(* IEC 61131-3 sources: SafePLC-Gen-Evaluation/Evaluation Results/eastman/run_03, 2 files *)

(* ---- io_declarations.st ---- *)
(* ==================================================  *)
(* PLC I/O Variable Declarations — CODESYS 3.5  *)
(* Generated by SafePLC-Gen Multimodal  *)
(* ==================================================  *)

VAR_GLOBAL
    (* --- Analog Inputs ---  *)
    FI_1_Raw                     AT %IW0       : INT := 0;    (* FI-1 — Flow indicator on feed line P-65 enterin  *)
    FI_2_Raw                     AT %IW2       : INT := 0;    (* FI-2 — Flow indicator on line P-54/P-53 associa  *)
    FI_3_Raw                     AT %IW4       : INT := 0;    (* FI-3 — Flow indicator on line P-57 associated w  *)
    TI_1_Raw                     AT %IW6       : INT := 0;    (* TI-1 — Temperature indicator TI-1, local panel   *)
    TI_4_Raw                     AT %IW8       : INT := 0;    (* TI-4 — Temperature indicator TI-4 on line P-12   *)
    TI_5_Raw                     AT %IW10      : INT := 0;    (* TI-5 — Temperature indicator TI-5 on line P-53   *)
    TI_6_Raw                     AT %IW12      : INT := 0;    (* TI-6 — Temperature indicator TI-6 on line assoc  *)
    TI_7_Raw                     AT %IW14      : INT := 0;    (* TI-7 — Temperature indicator TI-7 on line P-20/  *)
    TI_8_Raw                     AT %IW16      : INT := 0;    (* TI-8 — Temperature indicator TI-8 on line P-57   *)
    (* --- Analog Outputs ---  *)
    V_3_Out                      AT %QW0       : INT := 0;    (* V-3 — Control valve V-3 on line P-28 from Deca  *)
    V_4_Out                      AT %QW2       : INT := 0;    (* V-4 — Control valve V-4 on line P-74/P-12 feed  *)
    V_5_Out                      AT %QW4       : INT := 0;    (* V-5 — Control valve V-5 on line P-38/P-83 refl  *)
    V_7_Out                      AT %QW6       : INT := 0;    (* V-7 — Control valve V-7 on line P-19 vent or p  *)
END_VAR

(* ---- generated_code.st ---- *)
(* Generated by SafePLC-Gen Multimodal — CODESYS 3.5 *)
(* IEC 61131-3 Structured Text *)
(* Date: 2026-04-25T12:33:26.075096 *)

PROGRAM DistillationControl

VAR
    FI_1_Raw                     AT %IW0       : INT := 0;
    FI_2_Raw                     AT %IW2       : INT := 0;
    FI_3_Raw                     AT %IW4       : INT := 0;
    TI_1_Raw                     AT %IW6       : INT := 0;
    TI_4_Raw                     AT %IW8       : INT := 0;
    TI_5_Raw                     AT %IW10      : INT := 0;
    TI_6_Raw                     AT %IW12      : INT := 0;
    TI_7_Raw                     AT %IW14      : INT := 0;
    TI_8_Raw                     AT %IW16      : INT := 0;
    V_3_Out                      AT %QW0       : INT := 0;
    V_4_Out                      AT %QW2       : INT := 0;
    V_5_Out                      AT %QW4       : INT := 0;
    V_7_Out                      AT %QW6       : INT := 0;
END_VAR

VAR
    FirstScan                    : BOOL := TRUE;

    FI_1_Scaled                  : REAL := 0.0;
    FI_2_Scaled                  : REAL := 0.0;
    FI_3_Scaled                  : REAL := 0.0;
    TI_1_Scaled                  : REAL := 0.0;
    TI_4_Scaled                  : REAL := 0.0;
    TI_5_Scaled                  : REAL := 0.0;
    TI_6_Scaled                  : REAL := 0.0;
    TI_7_Scaled                  : REAL := 0.0;
    TI_8_Scaled                  : REAL := 0.0;

    FI_1_HH_SP                   : REAL := 180.0;
    FI_1_H_SP                    : REAL := 160.0;
    FI_1_L_SP                    : REAL := 40.0;
    FI_1_LL_SP                   : REAL := 20.0;
    FI_1_Deadband                : REAL := 2.0;
    FI_1_HH                      : BOOL := FALSE;
    FI_1_H                       : BOOL := FALSE;
    FI_1_L                       : BOOL := FALSE;
    FI_1_LL                      : BOOL := FALSE;
    FI_1_HH_Latch                : SR := (S1 := FALSE, R := FALSE);
    FI_1_LL_Latch                : SR := (S1 := FALSE, R := FALSE);
    FI_1_HH_Ack                  : BOOL := FALSE;
    FI_1_LL_Ack                  : BOOL := FALSE;

    FI_2_HH_SP                   : REAL := 180.0;
    FI_2_H_SP                    : REAL := 160.0;
    FI_2_L_SP                    : REAL := 40.0;
    FI_2_LL_SP                   : REAL := 20.0;
    FI_2_Deadband                : REAL := 2.0;
    FI_2_HH                      : BOOL := FALSE;
    FI_2_H                       : BOOL := FALSE;
    FI_2_L                       : BOOL := FALSE;
    FI_2_LL                      : BOOL := FALSE;
    FI_2_HH_Latch                : SR := (S1 := FALSE, R := FALSE);
    FI_2_LL_Latch                : SR := (S1 := FALSE, R := FALSE);
    FI_2_HH_Ack                  : BOOL := FALSE;
    FI_2_LL_Ack                  : BOOL := FALSE;

    FI_3_HH_SP                   : REAL := 180.0;
    FI_3_H_SP                    : REAL := 160.0;
    FI_3_L_SP                    : REAL := 40.0;
    FI_3_LL_SP                   : REAL := 20.0;
    FI_3_Deadband                : REAL := 2.0;
    FI_3_HH                      : BOOL := FALSE;
    FI_3_H                       : BOOL := FALSE;
    FI_3_L                       : BOOL := FALSE;
    FI_3_LL                      : BOOL := FALSE;
    FI_3_HH_Latch                : SR := (S1 := FALSE, R := FALSE);
    FI_3_LL_Latch                : SR := (S1 := FALSE, R := FALSE);
    FI_3_HH_Ack                  : BOOL := FALSE;
    FI_3_LL_Ack                  : BOOL := FALSE;

    TI_1_HH_SP                   : REAL := 120.0;
    TI_1_H_SP                    : REAL := 110.0;
    TI_1_L_SP                    : REAL := 30.0;
    TI_1_LL_SP                   : REAL := 20.0;
    TI_1_Deadband                : REAL := 1.0;
    TI_1_HH                      : BOOL := FALSE;
    TI_1_H                       : BOOL := FALSE;
    TI_1_L                       : BOOL := FALSE;
    TI_1_LL                      : BOOL := FALSE;
    TI_1_HH_Latch                : SR := (S1 := FALSE, R := FALSE);
    TI_1_LL_Latch                : SR := (S1 := FALSE, R := FALSE);
    TI_1_HH_Ack                  : BOOL := FALSE;
    TI_1_LL_Ack                  : BOOL := FALSE;

    TI_4_HH_SP                   : REAL := 120.0;
    TI_4_H_SP                    : REAL := 110.0;
    TI_4_L_SP                    : REAL := 30.0;
    TI_4_LL_SP                   : REAL := 20.0;
    TI_4_Deadband                : REAL := 1.0;
    TI_4_HH                      : BOOL := FALSE;
    TI_4_H                       : BOOL := FALSE;
    TI_4_L                       : BOOL := FALSE;
    TI_4_LL                      : BOOL := FALSE;
    TI_4_HH_Latch                : SR := (S1 := FALSE, R := FALSE);
    TI_4_LL_Latch                : SR := (S1 := FALSE, R := FALSE);
    TI_4_HH_Ack                  : BOOL := FALSE;
    TI_4_LL_Ack                  : BOOL := FALSE;

    TI_5_HH_SP                   : REAL := 120.0;
    TI_5_H_SP                    : REAL := 110.0;
    TI_5_L_SP                    : REAL := 30.0;
    TI_5_LL_SP                   : REAL := 20.0;
    TI_5_Deadband                : REAL := 1.0;
    TI_5_HH                      : BOOL := FALSE;
    TI_5_H                       : BOOL := FALSE;
    TI_5_L                       : BOOL := FALSE;
    TI_5_LL                      : BOOL := FALSE;
    TI_5_HH_Latch                : SR := (S1 := FALSE, R := FALSE);
    TI_5_LL_Latch                : SR := (S1 := FALSE, R := FALSE);
    TI_5_HH_Ack                  : BOOL := FALSE;
    TI_5_LL_Ack                  : BOOL := FALSE;

    TI_6_HH_SP                   : REAL := 120.0;
    TI_6_H_SP                    : REAL := 110.0;
    TI_6_L_SP                    : REAL := 30.0;
    TI_6_LL_SP                   : REAL := 20.0;
    TI_6_Deadband                : REAL := 1.0;
    TI_6_HH                      : BOOL := FALSE;
    TI_6_H                       : BOOL := FALSE;
    TI_6_L                       : BOOL := FALSE;
    TI_6_LL                      : BOOL := FALSE;
    TI_6_HH_Latch                : SR := (S1 := FALSE, R := FALSE);
    TI_6_LL_Latch                : SR := (S1 := FALSE, R := FALSE);
    TI_6_HH_Ack                  : BOOL := FALSE;
    TI_6_LL_Ack                  : BOOL := FALSE;

    TI_7_HH_SP                   : REAL := 120.0;
    TI_7_H_SP                    : REAL := 110.0;
    TI_7_L_SP                    : REAL := 30.0;
    TI_7_LL_SP                   : REAL := 20.0;
    TI_7_Deadband                : REAL := 1.0;
    TI_7_HH                      : BOOL := FALSE;
    TI_7_H                       : BOOL := FALSE;
    TI_7_L                       : BOOL := FALSE;
    TI_7_LL                      : BOOL := FALSE;
    TI_7_HH_Latch                : SR := (S1 := FALSE, R := FALSE);
    TI_7_LL_Latch                : SR := (S1 := FALSE, R := FALSE);
    TI_7_HH_Ack                  : BOOL := FALSE;
    TI_7_LL_Ack                  : BOOL := FALSE;

    TI_8_HH_SP                   : REAL := 120.0;
    TI_8_H_SP                    : REAL := 110.0;
    TI_8_L_SP                    : REAL := 30.0;
    TI_8_LL_SP                   : REAL := 20.0;
    TI_8_Deadband                : REAL := 1.0;
    TI_8_HH                      : BOOL := FALSE;
    TI_8_H                       : BOOL := FALSE;
    TI_8_L                       : BOOL := FALSE;
    TI_8_LL                      : BOOL := FALSE;
    TI_8_HH_Latch                : SR := (S1 := FALSE, R := FALSE);
    TI_8_LL_Latch                : SR := (S1 := FALSE, R := FALSE);
    TI_8_HH_Ack                  : BOOL := FALSE;
    TI_8_LL_Ack                  : BOOL := FALSE;

    V3_SP                        : REAL := 100.0;
    V3_Kp                        : REAL := 1.2;
    V3_Ki                        : REAL := 0.05;
    V3_Integral                  : REAL := 0.0;
    V3_Error                     : REAL := 0.0;
    V3_Output                    : REAL := 50.0;

    V4_SP                        : REAL := 80.0;
    V4_Kp                        : REAL := 1.5;
    V4_Ki                        : REAL := 0.04;
    V4_Integral                  : REAL := 0.0;
    V4_Error                     : REAL := 0.0;
    V4_Output                    : REAL := 50.0;

    V5_SP                        : REAL := 100.0;
    V5_Kp                        : REAL := 1.2;
    V5_Ki                        : REAL := 0.05;
    V5_Integral                  : REAL := 0.0;
    V5_Error                     : REAL := 0.0;
    V5_Output                    : REAL := 50.0;

    V7_SP                        : REAL := 100.0;
    V7_Kp                        : REAL := 1.2;
    V7_Ki                        : REAL := 0.05;
    V7_Integral                  : REAL := 0.0;
    V7_Error                     : REAL := 0.0;
    V7_Output                    : REAL := 50.0;

    System_Alarm                 : BOOL := FALSE;
END_VAR

IF FirstScan THEN
    V_3_Out     := 6554;
    V_4_Out     := 6554;
    V_5_Out     := 6554;
    V_7_Out     := 6554;
    V3_Integral := 0.0;
    V4_Integral := 0.0;
    V5_Integral := 0.0;
    V7_Integral := 0.0;
    FI_1_HH_Latch(S1 := FALSE, R := FALSE);
    FI_1_LL_Latch(S1 := FALSE, R := FALSE);
    FI_2_HH_Latch(S1 := FALSE, R := FALSE);
    FI_2_LL_Latch(S1 := FALSE, R := FALSE);
    FI_3_HH_Latch(S1 := FALSE, R := FALSE);
    FI_3_LL_Latch(S1 := FALSE, R := FALSE);
    TI_1_HH_Latch(S1 := FALSE, R := FALSE);
    TI_1_LL_Latch(S1 := FALSE, R := FALSE);
    TI_4_HH_Latch(S1 := FALSE, R := FALSE);
    TI_4_LL_Latch(S1 := FALSE, R := FALSE);
    TI_5_HH_Latch(S1 := FALSE, R := FALSE);
    TI_5_LL_Latch(S1 := FALSE, R := FALSE);
    TI_6_HH_Latch(S1 := FALSE, R := FALSE);
    TI_6_LL_Latch(S1 := FALSE, R := FALSE);
    TI_7_HH_Latch(S1 := FALSE, R := FALSE);
    TI_7_LL_Latch(S1 := FALSE, R := FALSE);
    TI_8_HH_Latch(S1 := FALSE, R := FALSE);
    TI_8_LL_Latch(S1 := FALSE, R := FALSE);
    FirstScan := FALSE;
    RETURN;
END_IF;

FI_1_Scaled := ((INT_TO_REAL(FI_1_Raw) - 6554.0) / (32767.0 - 6554.0)) * 200.0;
FI_2_Scaled := ((INT_TO_REAL(FI_2_Raw) - 6554.0) / (32767.0 - 6554.0)) * 200.0;
FI_3_Scaled := ((INT_TO_REAL(FI_3_Raw) - 6554.0) / (32767.0 - 6554.0)) * 200.0;
TI_1_Scaled := ((INT_TO_REAL(TI_1_Raw) - 6554.0) / (32767.0 - 6554.0)) * 150.0;
TI_4_Scaled := ((INT_TO_REAL(TI_4_Raw) - 6554.0) / (32767.0 - 6554.0)) * 150.0;
TI_5_Scaled := ((INT_TO_REAL(TI_5_Raw) - 6554.0) / (32767.0 - 6554.0)) * 150.0;
TI_6_Scaled := ((INT_TO_REAL(TI_6_Raw) - 6554.0) / (32767.0 - 6554.0)) * 150.0;
TI_7_Scaled := ((INT_TO_REAL(TI_7_Raw) - 6554.0) / (32767.0 - 6554.0)) * 150.0;
TI_8_Scaled := ((INT_TO_REAL(TI_8_Raw) - 6554.0) / (32767.0 - 6554.0)) * 150.0;

IF FI_1_Scaled >= FI_1_HH_SP THEN
    FI_1_HH_Latch.S1 := TRUE;
ELSIF FI_1_Scaled <= (FI_1_HH_SP - FI_1_Deadband) THEN
    FI_1_HH_Latch.S1 := FALSE;
END_IF;
FI_1_HH_Latch.R := FI_1_HH_Ack AND (FI_1_Scaled < FI_1_HH_SP);
FI_1_HH_Latch(S1 := FI_1_HH_Latch.S1, R := FI_1_HH_Latch.R);
FI_1_HH := FI_1_HH_Latch.Q1;

IF FI_1_Scaled >= FI_1_H_SP THEN
    FI_1_H := TRUE;
ELSIF FI_1_Scaled <= (FI_1_H_SP - FI_1_Deadband) THEN
    FI_1_H := FALSE;
END_IF;

IF FI_1_Scaled <= FI_1_L_SP THEN
    FI_1_L := TRUE;
ELSIF FI_1_Scaled >= (FI_1_L_SP + FI_1_Deadband) THEN
    FI_1_L := FALSE;
END_IF;

IF FI_1_Scaled <= FI_1_LL_SP THEN
    FI_1_LL_Latch.S1 := TRUE;
ELSIF FI_1_Scaled >= (FI_1_LL_SP + FI_1_Deadband) THEN
    FI_1_LL_Latch.S1 := FALSE;
END_IF;
FI_1_LL_Latch.R := FI_1_LL_Ack AND (FI_1_Scaled > FI_1_LL_SP);
FI_1_LL_Latch(S1 := FI_1_LL_Latch.S1, R := FI_1_LL_Latch.R);
FI_1_LL := FI_1_LL_Latch.Q1;

IF FI_2_Scaled >= FI_2_HH_SP THEN
    FI_2_HH_Latch.S1 := TRUE;
ELSIF FI_2_Scaled <= (FI_2_HH_SP - FI_2_Deadband) THEN
    FI_2_HH_Latch.S1 := FALSE;
END_IF;
FI_2_HH_Latch.R := FI_2_HH_Ack AND (FI_2_Scaled < FI_2_HH_SP);
FI_2_HH_Latch(S1 := FI_2_HH_Latch.S1, R := FI_2_HH_Latch.R);
FI_2_HH := FI_2_HH_Latch.Q1;

IF FI_2_Scaled >= FI_2_H_SP THEN
    FI_2_H := TRUE;
ELSIF FI_2_Scaled <= (FI_2_H_SP - FI_2_Deadband) THEN
    FI_2_H := FALSE;
END_IF;

IF FI_2_Scaled <= FI_2_L_SP THEN
    FI_2_L := TRUE;
ELSIF FI_2_Scaled >= (FI_2_L_SP + FI_2_Deadband) THEN
    FI_2_L := FALSE;
END_IF;

IF FI_2_Scaled <= FI_2_LL_SP THEN
    FI_2_LL_Latch.S1 := TRUE;
ELSIF FI_2_Scaled >= (FI_2_LL_SP + FI_2_Deadband) THEN
    FI_2_LL_Latch.S1 := FALSE;
END_IF;
FI_2_LL_Latch.R := FI_2_LL_Ack AND (FI_2_Scaled > FI_2_LL_SP);
FI_2_LL_Latch(S1 := FI_2_LL_Latch.S1, R := FI_2_LL_Latch.R);
FI_2_LL := FI_2_LL_Latch.Q1;

IF FI_3_Scaled >= FI_3_HH_SP THEN
    FI_3_HH_Latch.S1 := TRUE;
ELSIF FI_3_Scaled <= (FI_3_HH_SP - FI_3_Deadband) THEN
    FI_3_HH_Latch.S1 := FALSE;
END_IF;
FI_3_HH_Latch.R := FI_3_HH_Ack AND (FI_3_Scaled < FI_3_HH_SP);
FI_3_HH_Latch(S1 := FI_3_HH_Latch.S1, R := FI_3_HH_Latch.R);
FI_3_HH := FI_3_HH_Latch.Q1;

IF FI_3_Scaled >= FI_3_H_SP THEN
    FI_3_H := TRUE;
ELSIF FI_3_Scaled <= (FI_3_H_SP - FI_3_Deadband) THEN
    FI_3_H := FALSE;
END_IF;

IF FI_3_Scaled <= FI_3_L_SP THEN
    FI_3_L := TRUE;
ELSIF FI_3_Scaled >= (FI_3_L_SP + FI_3_Deadband) THEN
    FI_3_L := FALSE;
END_IF;

IF FI_3_Scaled <= FI_3_LL_SP THEN
    FI_3_LL_Latch.S1 := TRUE;
ELSIF FI_3_Scaled >= (FI_3_LL_SP + FI_3_Deadband) THEN
    FI_3_LL_Latch.S1 := FALSE;
END_IF;
FI_3_LL_Latch.R := FI_3_LL_Ack AND (FI_3_Scaled > FI_3_LL_SP);
FI_3_LL_Latch(S1 := FI_3_LL_Latch.S1, R := FI_3_LL_Latch.R);
FI_3_LL := FI_3_LL_Latch.Q1;

IF TI_1_Scaled >= TI_1_HH_SP THEN
    TI_1_HH_Latch.S1 := TRUE;
ELSIF TI_1_Scaled <= (TI_1_HH_SP - TI_1_Deadband) THEN
    TI_1_HH_Latch.S1 := FALSE;
END_IF;
TI_1_HH_Latch.R := TI_1_HH_Ack AND (TI_1_Scaled < TI_1_HH_SP);
TI_1_HH_Latch(S1 := TI_1_HH_Latch.S1, R := TI_1_HH_Latch.R);
TI_1_HH := TI_1_HH_Latch.Q1;

IF TI_1_Scaled >= TI_1_H_SP THEN
    TI_1_H := TRUE;
ELSIF TI_1_Scaled <= (TI_1_H_SP - TI_1_Deadband) THEN
    TI_1_H := FALSE;
END_IF;

IF TI_1_Scaled <= TI_1_L_SP THEN
    TI_1_L := TRUE;
ELSIF TI_1_Scaled >= (TI_1_L_SP + TI_1_Deadband) THEN
    TI_1_L := FALSE;
END_IF;

IF TI_1_Scaled <= TI_1_LL_SP THEN
    TI_1_LL_Latch.S1 := TRUE;
ELSIF TI_1_Scaled >= (TI_1_LL_SP + TI_1_Deadband) THEN
    TI_1_LL_Latch.S1 := FALSE;
END_IF;
TI_1_LL_Latch.R := TI_1_LL_Ack AND (TI_1_Scaled > TI_1_LL_SP);
TI_1_LL_Latch(S1 := TI_1_LL_Latch.S1, R := TI_1_LL_Latch.R);
TI_1_LL := TI_1_LL_Latch.Q1;

IF TI_4_Scaled >= TI_4_HH_SP THEN
    TI_4_HH_Latch.S1 := TRUE;
ELSIF TI_4_Scaled <= (TI_4_HH_SP - TI_4_Deadband) THEN
    TI_4_HH_Latch.S1 := FALSE;
END_IF;
TI_4_HH_Latch.R := TI_4_HH_Ack AND (TI_4_Scaled < TI_4_HH_SP);
TI_4_HH_Latch(S1 := TI_4_HH_Latch.S1, R := TI_4_HH_Latch.R);
TI_4_HH := TI_4_HH_Latch.Q1;

IF TI_4_Scaled >= TI_4_H_SP THEN
    TI_4_H := TRUE;
ELSIF TI_4_Scaled <= (TI_4_H_SP - TI_4_Deadband) THEN
    TI_4_H := FALSE;
END_IF;

IF TI_4_Scaled <= TI_4_L_SP THEN
    TI_4_L := TRUE;
ELSIF TI_4_Scaled >= (TI_4_L_SP + TI_4_Deadband) THEN
    TI_4_L := FALSE;
END_IF;

IF TI_4_Scaled <= TI_4_LL_SP THEN
    TI_4_LL_Latch.S1 := TRUE;
ELSIF TI_4_Scaled >= (TI_4_LL_SP + TI_4_Deadband) THEN
    TI_4_LL_Latch.S1 := FALSE;
END_IF;
TI_4_LL_Latch.R := TI_4_LL_Ack AND (TI_4_Scaled > TI_4_LL_SP);
TI_4_LL_Latch(S1 := TI_4_LL_Latch.S1, R := TI_4_LL_Latch.R);
TI_4_LL := TI_4_LL_Latch.Q1;

IF TI_5_Scaled >= TI_5_HH_SP THEN
    TI_5_HH_Latch.S1 := TRUE;
ELSIF TI_5_Scaled <= (TI_5_HH_SP - TI_5_Deadband) THEN
    TI_5_HH_Latch.S1 := FALSE;
END_IF;
TI_5_HH_Latch.R := TI_5_HH_Ack AND (TI_5_Scaled < TI_5_HH_SP);
TI_5_HH_Latch(S1 := TI_5_HH_Latch.S1, R := TI_5_HH_Latch.R);
TI_5_HH := TI_5_HH_Latch.Q1;

IF TI_5_Scaled >= TI_5_H_SP THEN
    TI_5_H := TRUE;
ELSIF TI_5_Scaled <= (TI_5_H_SP - TI_5_Deadband) THEN
    TI_5_H := FALSE;
END_IF;

IF TI_5_Scaled <= TI_5_L_SP THEN
    TI_5_L := TRUE;
ELSIF TI_5_Scaled >= (TI_5_L_SP + TI_5_Deadband) THEN
    TI_5_L := FALSE;
END_IF;

IF TI_5_Scaled <= TI_5_LL_SP THEN
    TI_5_LL_Latch.S1 := TRUE;
ELSIF TI_5_Scaled >= (TI_5_LL_SP + TI_5_Deadband) THEN
    TI_5_LL_Latch.S1 := FALSE;
END_IF;
TI_5_LL_Latch.R := TI_5_LL_Ack AND (TI_5_Scaled > TI_5_LL_SP);
TI_5_LL_Latch(S1 := TI_5_LL_Latch.S1, R := TI_5_LL_Latch.R);
TI_5_LL := TI_5_LL_Latch.Q1;

IF TI_6_Scaled >= TI_6_HH_SP THEN
    TI_6_HH_Latch.S1 := TRUE;
ELSIF TI_6_Scaled <= (TI_6_HH_SP - TI_6_Deadband) THEN
    TI_6_HH_Latch.S1 := FALSE;
END_IF;
TI_6_HH_Latch.R := TI_6_HH_Ack AND (TI_6_Scaled < TI_6_HH_SP);
TI_6_HH_Latch(S1 := TI_6_HH_Latch.S1, R := TI_6_HH_Latch.R);
TI_6_HH := TI_6_HH_Latch.Q1;

IF TI_6_Scaled >= TI_6_H_SP THEN
    TI_6_H := TRUE;
ELSIF TI_6_Scaled <= (TI_6_H_SP - TI_6_Deadband) THEN
    TI_6_H := FALSE;
END_IF;

IF TI_6_Scaled <= TI_6_L_SP THEN
    TI_6_L := TRUE;
ELSIF TI_6_Scaled >= (TI_6_L_SP + TI_6_Deadband) THEN
    TI_6_L := FALSE;
END_IF;

IF TI_6_Scaled <= TI_6_LL_SP THEN
    TI_6_LL_Latch.S1 := TRUE;
ELSIF TI_6_Scaled >= (TI_6_LL_SP + TI_6_Deadband) THEN
    TI_6_LL_Latch.S1 := FALSE;
END_IF;
TI_6_LL_Latch.R := TI_6_LL_Ack AND (TI_6_Scaled > TI_6_LL_SP);
TI_6_LL_Latch(S1 := TI_6_LL_Latch.S1, R := TI_6_LL_Latch.R);
TI_6_LL := TI_6_LL_Latch.Q1;

IF TI_7_Scaled >= TI_7_HH_SP THEN
    TI_7_HH_Latch.S1 := TRUE;
ELSIF TI_7_Scaled <= (TI_7_HH_SP - TI_7_Deadband) THEN
    TI_7_HH_Latch.S1 := FALSE;
END_IF;
TI_7_HH_Latch.R := TI_7_HH_Ack AND (TI_7_Scaled < TI_7_HH_SP);
TI_7_HH_Latch(S1 := TI_7_HH_Latch.S1, R := TI_7_HH_Latch.R);
TI_7_HH := TI_7_HH_Latch.Q1;

IF TI_7_Scaled >= TI_7_H_SP THEN
    TI_7_H := TRUE;
ELSIF TI_7_Scaled <= (TI_7_H_SP - TI_7_Deadband) THEN
    TI_7_H := FALSE;
END_IF;

IF TI_7_Scaled <= TI_7_L_SP THEN
    TI_7_L := TRUE;
ELSIF TI_7_Scaled >= (TI_7_L_SP + TI_7_Deadband) THEN
    TI_7_L := FALSE;
END_IF;

IF TI_7_Scaled <= TI_7_LL_SP THEN
    TI_7_LL_Latch.S1 := TRUE;
ELSIF TI_7_Scaled >= (TI_7_LL_SP + TI_7_Deadband) THEN
    TI_7_LL_Latch.S1 := FALSE;
END_IF;
TI_7_LL_Latch.R := TI_7_LL_Ack AND (TI_7_Scaled > TI_7_LL_SP);
TI_7_LL_Latch(S1 := TI_7_LL_Latch.S1, R := TI_7_LL_Latch.R);
TI_7_LL := TI_7_LL_Latch.Q1;

IF TI_8_Scaled >= TI_8_HH_SP THEN
    TI_8_HH_Latch.S1 := TRUE;
ELSIF TI_8_Scaled <= (TI_8_HH_SP - TI_8_Deadband) THEN
    TI_8_HH_Latch.S1 := FALSE;
END_IF;
TI_8_HH_Latch.R := TI_8_HH_Ack AND (TI_8_Scaled < TI_8_HH_SP);
TI_8_HH_Latch(S1 := TI_8_HH_Latch.S1, R := TI_8_HH_Latch.R);
TI_8_HH := TI_8_HH_Latch.Q1;

IF TI_8_Scaled >= TI_8_H_SP THEN
    TI_8_H := TRUE;
ELSIF TI_8_Scaled <= (TI_8_H_SP - TI_8_Deadband) THEN
    TI_8_H := FALSE;
END_IF;

IF TI_8_Scaled <= TI_8_L_SP THEN
    TI_8_L := TRUE;
ELSIF TI_8_Scaled >= (TI_8_L_SP + TI_8_Deadband) THEN
    TI_8_L := FALSE;
END_IF;

IF TI_8_Scaled <= TI_8_LL_SP THEN
    TI_8_LL_Latch.S1 := TRUE;
ELSIF TI_8_Scaled >= (TI_8_LL_SP + TI_8_Deadband) THEN
    TI_8_LL_Latch.S1 := FALSE;
END_IF;
TI_8_LL_Latch.R := TI_8_LL_Ack AND (TI_8_Scaled > TI_8_LL_SP);
TI_8_LL_Latch(S1 := TI_8_LL_Latch.S1, R := TI_8_LL_Latch.R);
TI_8_LL := TI_8_LL_Latch.Q1;

V7_Error    := V7_SP - FI_1_Scaled;
V7_Integral := V7_Integral + (V7_Ki * V7_Error);
IF V7_Integral > 100.0 THEN
    V7_Integral := 100.0;
ELSIF V7_Integral < 0.0 THEN
    V7_Integral := 0.0;
END_IF;
V7_Output := (V7_Kp * V7_Error) + V7_Integral;
IF V7_Output > 100.0 THEN
    V7_Output := 100.0;
ELSIF V7_Output < 0.0 THEN
    V7_Output := 0.0;
END_IF;
V_7_Out := REAL_TO_INT(6554.0 + (V7_Output / 100.0) * (32767.0 - 6554.0));

V5_Error    := V5_SP - FI_2_Scaled;
V5_Integral := V5_Integral + (V5_Ki * V5_Error);
IF V5_Integral > 100.0 THEN
    V5_Integral := 100.0;
ELSIF V5_Integral < 0.0 THEN
    V5_Integral := 0.0;
END_IF;
V5_Output := (V5_Kp * V5_Error) + V5_Integral;
IF V5_Output > 100.0 THEN
    V5_Output := 100.0;
ELSIF V5_Output < 0.0 THEN
    V5_Output := 0.0;
END_IF;
V_5_Out := REAL_TO_INT(6554.0 + (V5_Output / 100.0) * (32767.0 - 6554.0));

V3_Error    := V3_SP - FI_3_Scaled;
V3_Integral := V3_Integral + (V3_Ki * V3_Error);
IF V3_Integral > 100.0 THEN
    V3_Integral := 100.0;
ELSIF V3_Integral < 0.0 THEN
    V3_Integral := 0.0;
END_IF;
V3_Output := (V3_Kp * V3_Error) + V3_Integral;
IF V3_Output > 100.0 THEN
    V3_Output := 100.0;
ELSIF V3_Output < 0.0 THEN
    V3_Output := 0.0;
END_IF;
V_3_Out := REAL_TO_INT(6554.0 + (V3_Output / 100.0) * (32767.0 - 6554.0));

V4_Error    := V4_SP - TI_4_Scaled;
V4_Integral := V4_Integral + (V4_Ki * V4_Error);
IF V4_Integral > 100.0 THEN
    V4_Integral := 100.0;
ELSIF V4_Integral < 0.0 THEN
    V4_Integral := 0.0;
END_IF;
V4_Output := (V4_Kp * V4_Error) + V4_Integral;
IF V4_Output > 100.0 THEN
    V4_Output := 100.0;
ELSIF V4_Output < 0.0 THEN
    V4_Output := 0.0;
END_IF;
V_4_Out := REAL_TO_INT(6554.0 + (V4_Output / 100.0) * (32767.0 - 6554.0));

System_Alarm :=
    FI_1_HH_Latch.Q1 OR FI_1_LL_Latch.Q1 OR FI_1_H OR FI_1_L OR
    FI_2_HH_Latch.Q1 OR FI_2_LL_Latch.Q1 OR FI_2_H OR FI_2_L OR
    FI_3_HH_Latch.Q1 OR FI_3_LL_Latch.Q1 OR FI_3_H OR FI_3_L OR
    TI_1_HH_Latch.Q1 OR TI_1_LL_Latch.Q1 OR TI_1_H OR TI_1_L OR
    TI_4_HH_Latch.Q1 OR TI_4_LL_Latch.Q1 OR TI_4_H OR TI_4_L OR
    TI_5_HH_Latch.Q1 OR TI_5_LL_Latch.Q1 OR TI_5_H OR TI_5_L OR
    TI_6_HH_Latch.Q1 OR TI_6_LL_Latch.Q1 OR TI_6_H OR TI_6_L OR
    TI_7_HH_Latch.Q1 OR TI_7_LL_Latch.Q1 OR TI_7_H OR TI_7_L OR
    TI_8_HH_Latch.Q1 OR TI_8_LL_Latch.Q1 OR TI_8_H OR TI_8_L;

END_PROGRAM
